PROGRAM prg_MotorMetDrukknop
VAR
  	T1: R_TRIG;
	Drukknop		AT		%I*		:BOOL;
	Hoofdschakelaar	AT		%I*		:BOOL;
	
	MotorLinks		AT		%Q*		:BOOL;
	MotorRechts		AT		%Q*		:BOOL;

	Switch: BOOL;
END_VAR

T1(CLK := Drukknop);

IF Hoofdschakelaar AND T1.Q THEN
    IF MotorLinks OR MotorRechts THEN
        MotorLinks := FALSE;
        MotorRechts := FALSE;
        Switch := NOT Switch;
    ELSIF NOT Switch THEN
        MotorLinks := TRUE;
    ELSE
        MotorRechts := TRUE;
    END_IF
END_IF

END_PROGRAM

(* stored: Version 1.1.0.1, ProductVersion 3.1.4024.15
   POU prg_MotorMetDrukknop: Id {7270e293-eb2f-4d69-a11e-ba48b35146ec}, SpecialFunc None *)
